FUNCTION_BLOCK FB_Pulse
VAR_INPUT
END_VAR
VAR_OUTPUT
END_VAR
VAR
END_VAR

END_FUNCTION_BLOCK

(* stored: Version 1.1.0.1, ProductVersion 3.1.4024.13
   POU FB_Pulse: Id {9c76488e-ebf0-4cd6-90f0-9b7593e60c6d}, SpecialFunc None *)
